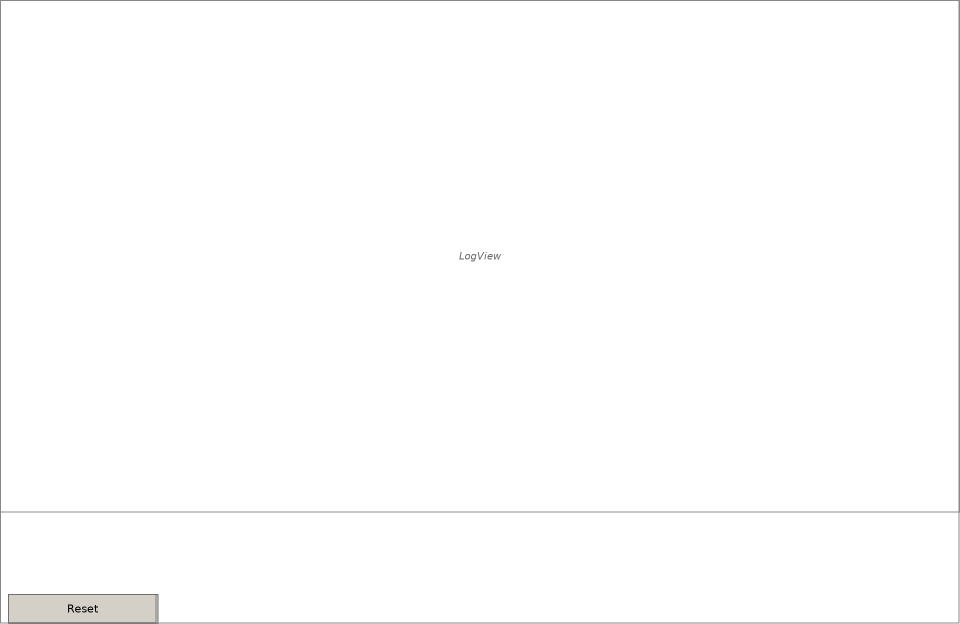
VISUALIZATION VISU_TEST_LOGVIEW  // 960x624
    Frame (0,0 960x512)
        shows LogView(fbLogView := PRG_TEST_LOGVIEW.fbLogView)
    Button (8,594 150x30), "Reset"
        tap PRG_TEST_LOGVIEW.fbLogView.bReset
END_VISUALIZATION

(* stored: Version 1.1.0.1, ProductVersion 3.1.4024.11
   Visu VISU_TEST_LOGVIEW: Id {3f5379d1-b9c7-4625-a2ba-573d75c78488} *)
